// TwinCAT 3 PLC project FncStructPlc
// ProgramVersion: 3.1.4024.0
// libraries:
//   Tc2_Standard, * (Beckhoff Automation GmbH)
//   Tc2_System, * (Beckhoff Automation GmbH)
//   Tc2_Utilities, * (Beckhoff Automation GmbH)
//   Tc3_Module, * (Beckhoff Automation GmbH)
// project tree:
//   DUTs/ E_EventType.TcDUT, ST_Event.TcDUT
//   / PlcTask.TcTTO
//   POUs/ Greater_Smaller.TcPOU, MAIN.TcPOU, UpdateEventTimestampWithSystemTime.TcPOU

CONFIGURATION FncStructPlc
    RESOURCE PLC ON TwinCAT3
        TASK PlcTask(INTERVAL := T#10ms, PRIORITY := 20);
        PROGRAM MAIN WITH PlcTask : MAIN;
    END_RESOURCE
END_CONFIGURATION

// ---- DUTs/E_EventType.TcDUT
{attribute 'qualified_only'}
{attribute 'strict'}
TYPE E_EventType :
(
	Alarm := 0,
	Message := 1
);
END_TYPE

// ---- DUTs/ST_Event.TcDUT
TYPE ST_Event :
STRUCT
	eEventType : E_EventType;
	eEventSeverity : TcEventSeverity;
	nEventIdentity : UDINT;
	sEventText : STRING(255);
	dtTimeStamp : DATE_AND_TIME;
END_STRUCT
END_TYPE

// ---- POUs/MAIN.TcPOU
PROGRAM MAIN
VAR
	aEvent : ARRAY[1..100] OF ST_Event;
	sTempString : STRING(255);
	
	nReturnGreater : INT;
	nReturnSmaller : INT;
	
	UpdateEventTimestam : ST_Event;
	aBoolean : BOOL := FALSE;
END_VAR

IF NOT aBoolean THEN
	sTempString := aEvent[33].sEventText;
	
	Greater_Smaller(nNumber1 := 8,
		nNumber2 := 15,
		nGreater => nReturnGreater,
		nSmaller => nReturnSmaller);
		
	UpdateEventTimestampWithSystemTime(stEvent := UpdateEventTimestam);
	aBoolean := TRUE;
END_IF

END_PROGRAM

// ---- POUs/Greater_Smaller.TcPOU
FUNCTION Greater_Smaller
VAR_INPUT
	nNumber1 : INT;
	nNumber2 : INT;
END_VAR
VAR_OUTPUT
	nGreater : INT;
	nSmaller : INT;
END_VAR

IF nNumber1 > nNumber2 THEN
	nGreater := nNumber1;
	nSmaller := nNumber2;
ELSE
	nGreater := nNumber2;
	nSmaller := nNumber1;	
END_IF

END_FUNCTION

// ---- POUs/UpdateEventTimestampWithSystemTime.TcPOU
FUNCTION UpdateEventTimestampWithSystemTime
VAR_INPUT
	stEvent : REFERENCE TO ST_Event;
END_VAR
VAR
	fbGETSYSTEMTIME : GETSYSTEMTIME;
	stFileName : T_FILETIME;
END_VAR

fbGETSYSTEMTIME(timeLoDW=>stFileName.dwLowDateTime,
 timeHiDW => stFileName.dwHighDateTime);
 
stEvent.dtTimeStamp := FILETIME_TO_DT(fileTime := stFileName);

END_FUNCTION
